Universal Robots PolyScope program: test2.urp

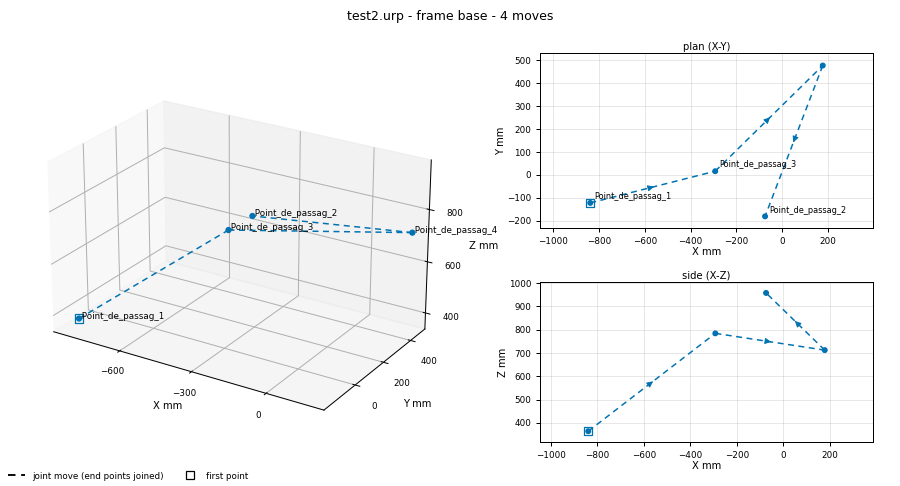
[picture p0: tool path of test2.urp in frame base, 4 of 4 moves have a stored position in this frame; points joined in program order, loops and branches not executed]
ProgramRoot directory=/programs; kinematics=(a=[0, -0.425, -0.39225, 0, 0, 0], d=[0.08916, 0, 0, 0.10915, 0.09465, 0.0823], alpha=[1.5708, 0, 0, 1.5708, -1.5708, 0], deltaTheta=[0, 0, 0, 0, 0, 0], status=notInitialized); name=test2; programVersion=(project__name=PolyScope, major__version=1, minor__version=6, svn__revision=9671, build__date=Dec 17 2012, 15:17:18); robotEnvironmentFileName=default
  MainProgram cartesianAcceleration=1.2; cartesianSpeed=0.25; jointAcceleration=1.3962634015954636; jointSpeed=1.0471975511965976; moveAsFastAsPossible=true; sharedProcessMoveBlendRadius=0.025; featureReference=(installationNameReference=Base); motionType=JOINT_SPACE
    Action analogValue=4.0; digitalValue=0; payloadValue=0.0; selectedAnalogSensor=-1; selectedDigitalSensor=-1; type=NO_ACTION
    Move cartesianAcceleration=1.2; cartesianSpeed=0.25; jointAcceleration=1.3962634015954636; jointSpeed=1.0471975511965976; moveAsFastAsPossible=true; sharedProcessMoveBlendRadius=0.025; featureReference=(installationNameReference=Base); motionType=JOINT_SPACE
      Waypoint blendRadius=0.05; cartesianAcceleration=1.2; cartesianSpeed=0.25; jointAcceleration=1.3962634015954636; jointSpeed=1.0471975511965976; nextMotionTime=2.0; stoppoint=true; useSharedBlendParameter=true; useSharedParameters=true; position=TCP in base x=-838.509 y=-122.401 z=364.333 mm, rx=1.8158 ry=-0.705 rz=0.5545 rad; joints [-4.392, -23.429, -1.27, -46.523, -20.467, 114.949] deg; positionType=FIXED_POSITION; waypointPoseInFeatureCoordinates=(pos=(x=-0.8385093780549049, y=-0.12240143348759339, z=0.3643331878433284), rot=(x=1.815762511318024, y=-0.7049557056024709, z=0.5545232373885608)); name=Point_de_passag_1
      Waypoint blendRadius=0.05; cartesianAcceleration=1.2; cartesianSpeed=0.25; jointAcceleration=1.3962634015954636; jointSpeed=1.0471975511965976; nextMotionTime=2.0; stoppoint=true; useSharedBlendParameter=true; useSharedParameters=true; position=TCP in base x=-292.638 y=16.165 z=784.549 mm, rx=1.6259 ry=-1.0494 rz=-0.252 rad; joints [-42.623, -54.341, -53.074, 14.688, -20.43, 114.949] deg; positionType=FIXED_POSITION; waypointPoseInFeatureCoordinates=(pos=(x=-0.29263753177219703, y=0.016164581038863132, z=0.7845485171083324), rot=(x=1.6258858774871885, y=-1.049376980538497, z=-0.2519872603528668)); name=Point_de_passag_3
      Waypoint blendRadius=0.05; cartesianAcceleration=1.2; cartesianSpeed=0.25; jointAcceleration=1.3962634015954636; jointSpeed=1.0471975511965976; nextMotionTime=2.0; stoppoint=true; useSharedBlendParameter=true; useSharedParameters=true; position=TCP in base x=177.195 y=477.816 z=712.499 mm, rx=0.4876 ry=-1.0644 rz=-1.7821 rad; joints [-130.755, -22.803, -66.546, -14.169, 33.597, 114.949] deg; positionType=FIXED_POSITION; waypointPoseInFeatureCoordinates=(pos=(x=0.17719493512549203, y=0.4778159234633474, z=0.7124986989936754), rot=(x=0.4875502965812094, y=-1.0643874836156988, z=-1.7821084481574563)); name=Point_de_passag_4
    Action analogValue=4.0; digitalValue=0; payloadValue=0.0; selectedAnalogSensor=-1; selectedDigitalSensor=-1; type=NO_ACTION
    Move cartesianAcceleration=1.2; cartesianSpeed=0.25; jointAcceleration=1.3962634015954636; jointSpeed=1.0471975511965976; moveAsFastAsPossible=true; sharedProcessMoveBlendRadius=0.025; featureReference=(installationNameReference=Base); motionType=JOINT_SPACE
      Waypoint blendRadius=0.05; cartesianAcceleration=1.2; cartesianSpeed=0.25; jointAcceleration=1.3962634015954636; jointSpeed=1.0471975511965976; nextMotionTime=2.0; stoppoint=true; useSharedBlendParameter=true; useSharedParameters=true; position=TCP in base x=-74.824 y=-181.074 z=958.095 mm, rx=1.838 ry=0.0886 rz=-0.5633 rad; joints [-4.377, -91.181, -0.95, -46.523, -20.464, 114.949] deg; positionType=FIXED_POSITION; waypointPoseInFeatureCoordinates=(pos=(x=-0.07482391990537016, y=-0.1810740559227427, z=0.958095462548447), rot=(x=1.8380151952185702, y=0.08861910148715743, z=-0.5633295740156234)); name=Point_de_passag_2
